// LS Electric XG5000 project: carnactest
// PLC NewPLC

PROGRAM NewProgram (task: 스캔 프로그램)

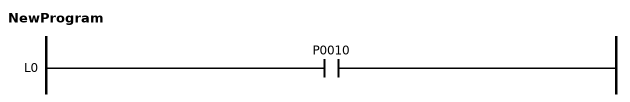
; L0
LOAD      P0010